{attribute 'qualified_only'}
{attribute 'strict'}
TYPE ePistonStatus :
(
	OPENED:=0,CLOSED,OPENING,CLOSING,ERROR,PAUSE
);
END_TYPE

(* stored: Version 1.1.0.1, ProductVersion 3.1.4024.12
   DUT ePistonStatus: Id {e467826b-7960-408b-9608-9daa829dc831} *)
